PROGRAM P_StationOpenLock
VAR
	_station:					REFERence TO ST_SystemStation;
	_bEnable: 					BOOL;
	_OpenLockCheck0FTrig:       Tc2_Standard.F_TRIG;
END_VAR

_station REF= G_arrStation[E_Station.OpenLock];
_station.arrName[E_Language.Chinese]:="解锁站";
_station.arrName[E_Language.Vietnamese]:="Mở khóa nhà ga";
_bEnable:=NOT GVL.stSetting.arrStationShield[E_Station.OpenLock];

IF GVL_Data.stRecipe.eMachineType=E_MachineType._311 THEN
	A_Home311();
	A_Auto311();
ELSE
	A_Home();
	A_Auto();
END_IF

_OpenLockCheck0FTrig(CLK:= GVL.I.bOpenLockCheck0, Q=> );

GVL._arrAutoTimer[E_Timer.SteeringCheck1F](IN:=NOT GVL.I.bSteeringCheck1 AND GVL.I.bSteeringAcquireElevator_Cyl_H, PT:=TO_TIME(GVL_Data.stRecipe.arrAutoTon[E_Timer.SteeringCheck1F]), Q=>GVL._arrAutoTimerOut[E_Timer.SteeringCheck1F] , ET=> );

ACTION A_Auto:
CASE _station.iStepNow OF
	1000:
		_station.arrInfo[E_Language.Chinese]:="初始化完成等待启动";
		IF _bEnable THEN
			_station.iStepNext:=1101;
		END_IF
	1101:
		_station.arrInfo[E_Language.Chinese]:="判断是否有料";
		IF NOT GVL.I.bOpenLockCheck THEN
			_station.iStepNext:=1201;
		END_IF
	1201:
		_station.arrInfo[E_Language.Chinese]:="请求上料";
		GVL.stHandshake.bOpenToSteering:=TRUE;
		IF GVL.stHandshake.bSteeringToOpen THEN
			_station.iStepNext:=1301;
		END_IF
	1301:
		_station.arrInfo[E_Language.Chinese]:="等待产品从旋转站流出";
		GVL.stOverTime.bOpenLockCheck:=TRUE;
		IF GVL._arrAutoTimerOut[E_Timer.SteeringCheck1F] THEN
			GVL.stOverTime.bOpenLockCheck:=FALSE;
			_station.iStepNext:=1401;//解锁站流入传感器安装后改为 1311
		END_IF
	1311:		
		_station.arrInfo[E_Language.Chinese]:="产品从旋转站流出确认";
		IF _OpenLockCheck0FTrig.Q THEN
			_station.iStepNext:=1401;
		END_IF	
	1401:
		_station.arrInfo[E_Language.Chinese]:="复位上料请求";
		GVL.stHandshake.bOpenToSteering:=FALSE;
		IF  NOT GVL.stHandshake.bSteeringToOpen THEN
			_station.iStepNext:=1411;
		END_IF
	1411:
		_station.arrInfo[E_Language.Chinese]:="等待产品到位";
		GVL.stOverTime.bOpenLockCheck:=TRUE;
		IF GVL.I.bOpenLockCheck THEN
			GVL.stOverTime.bOpenLockCheck:=FALSE;
			_station.iStepNext:=1501;
		END_IF			
	1501:
		_station.arrInfo[E_Language.Chinese]:="顶升气缸伸出";
		IF G_arrFbCylinder[E_Cylinder.OpenLockLift].M_WorkRequest() THEN
			IF GVL_Data.stRecipe.eMachineType=E_MachineType._373 AND NOT GVL.stSetting.bOpenLockPressShield THEN 
				_station.iStepNext:=1511;
			ELSE
			_station.iStepNext:=1601;
			END_IF
		END_IF
	1511:	
		_station.arrInfo[E_Language.Chinese]:="解压侧推气缸伸出";	
		IF G_arrFbCylinder[E_Cylinder.OpenLockPressPush].M_WorkRequest() THEN
			_station.iStepNext:=1521;
		END_IF
	1521:	
		_station.arrInfo[E_Language.Chinese]:="解压旋转气缸旋转";	
		IF G_arrFbCylinder[E_Cylinder.OpenLockPressRotate].M_WorkRequest() THEN
			_station.iStepNext:=1531;
		END_IF	
	1531:	
		_station.arrInfo[E_Language.Chinese]:="解压旋转气缸返回";	
		IF G_arrFbCylinder[E_Cylinder.OpenLockPressRotate].M_HomeRequest() THEN
			_station.iStepNext:=1541;		
		END_IF		
	1541:
		_station.arrInfo[E_Language.Chinese]:="解压侧推气缸缩回 侧推气缸伸出";
		IF M_PushWork() AND G_arrFbCylinder[E_Cylinder.OpenLockPressPush].M_HomeRequest() THEN
			_station.iStepNext:=1701;
		END_IF		
	1601:
		_station.arrInfo[E_Language.Chinese]:="侧推气缸伸出";
		IF M_PushWork() THEN
			_station.iStepNext:=1701;
		END_IF
	1701:
		_station.arrInfo[E_Language.Chinese]:="旋转气缸至右位 校平气缸伸出";
		IF G_arrFbCylinder[E_Cylinder.OpenLockRotate].M_WorkRequest() AND M_StandardWork() THEN
			_station.iStepNext:=1801;
		END_IF
	1801:
		_station.arrInfo[E_Language.Chinese]:="侧推气缸缩回 校平气缸缩回 阻挡气缸缩回";
		IF M_PushHome() AND M_StandardHome()  AND  G_arrFbCylinder[E_Cylinder.OpenLockPrevent].M_HomeRequest() THEN
           _station.iStepNext:=2001;
		END_IF
	2001:
		_station.arrInfo[E_Language.Chinese]:="等待取Uc站请求放料";
		IF GVL.stHandshake.bTakeUcToOpen THEN
			GVL.stHandshake.bOpenToTakeUc:=TRUE;
			GVL.stHandshake.bOpenToSteering:=TRUE;//同时请求旋转站放料
			_station.iStepNext:=2101;
		END_IF
	2101:
	     _station.arrInfo[E_Language.Chinese]:="顶升气缸下降,解锁旋转气缸至左位";
		IF G_arrFbCylinder[E_Cylinder.OpenLockLift].M_HomeRequest() AND G_arrFbCylinder[E_Cylinder.OpenLockRotate].M_HomeRequest() THEN
			_station.iStepNext:=2201;
		END_IF
	2201:
		_station.arrInfo[E_Language.Chinese]:="等待复位请求信号";
		IF NOT GVL.stHandshake.bTakeUcToOpen THEN
			GVL.stHandshake.bOpenToTakeUc:=FALSE;
			_station.iStepNext:=2301;
		END_IF		
	2301:
		_station.arrInfo[E_Language.Chinese]:="阻挡气缸伸出";
		IF G_arrFbCylinder[E_Cylinder.OpenLockPrevent].M_WorkRequest() THEN
			_station.iStepNext:=1201;
		END_IF		

END_CASE
END_ACTION

ACTION A_Auto311:
CASE _station.iStepNow OF
	1000:
		_station.arrInfo[E_Language.Chinese]:="初始化完成等待启动";
		IF _bEnable THEN
			_station.iStepNext:=1101;
		END_IF
	1101:
		_station.arrInfo[E_Language.Chinese]:="判断是否有料";
		IF NOT GVL.I.bOpenLockCheck THEN
			_station.iStepNext:=1201;
		END_IF
	1201:
		_station.arrInfo[E_Language.Chinese]:="请求上料";
		GVL.stHandshake.bOpenToSteering:=TRUE;
		IF GVL.stHandshake.bSteeringToOpen THEN
			_station.iStepNext:=1301;
		END_IF
	1301:
		_station.arrInfo[E_Language.Chinese]:="等待产品从旋转站流出";
		GVL.stOverTime.bOpenLockCheck:=TRUE;
		IF GVL._arrAutoTimerOut[E_Timer.SteeringCheck1F] THEN
			GVL.stOverTime.bOpenLockCheck:=FALSE;
			_station.iStepNext:=1401;//传感器安装后改为 1311
		END_IF
	1311:		
		_station.arrInfo[E_Language.Chinese]:="产品从旋转站流出确认";
		IF _OpenLockCheck0FTrig.Q THEN
			_station.iStepNext:=1401;
		END_IF			
	1401:
		_station.arrInfo[E_Language.Chinese]:="复位上料请求";
		GVL.stHandshake.bOpenToSteering:=FALSE;
		IF  NOT GVL.stHandshake.bSteeringToOpen THEN
			_station.iStepNext:=1411;
		END_IF
	1411:
		_station.arrInfo[E_Language.Chinese]:="等待产品到位";
		GVL.stOverTime.bOpenLockCheck:=TRUE;
		IF GVL.I.bOpenLockCheck THEN
			GVL.stOverTime.bOpenLockCheck:=FALSE;
			_station.iStepNext:=1501;
		END_IF			
	1501:
		_station.arrInfo[E_Language.Chinese]:="顶升气缸伸出";
		IF G_arrFbCylinder[E_Cylinder.OpenLockLift].M_WorkRequest() THEN
			_station.iStepNext:=1511;
		END_IF
	1511:		
		_station.arrInfo[E_Language.Chinese]:="检测工装有无误合盖";
		IF GVL.I.bFrockCloseCheck OR GVL.stSetting.bFrockCloseCheckShield THEN
			_station.iStepNext:=1601;
		ELSE
			_station.iStepNext:=1521;
		END_IF
	1521:	
		_station.arrInfo[E_Language.Chinese]:="置位工装检测失败记忆";
		GVL.TakeUcSafeCheckNG_OpenLock:=TRUE;
		IF GVL.TakeUcSafeCheckNG_OpenLock THEN
			_station.iStepNext:=2001;
		END_IF		
	1601:
		_station.arrInfo[E_Language.Chinese]:="升降气缸缩回";
		GVL.TakeUcSafeCheckNG_OpenLock:=FALSE;
		IF G_arrFbCylinder[E_Cylinder.OpenLockElevator].M_HomeRequest() THEN
			_station.iStepNext:=1701;
		END_IF
	1701:
		_station.arrInfo[E_Language.Chinese]:="按压气缸伸出";
		IF G_arrFbCylinder[E_Cylinder.OpenLockPin].M_WorkRequest() THEN
			_station.iStepNext:=1801;
		END_IF
	1801:
		_station.arrInfo[E_Language.Chinese]:="平移气缸缩回";
		IF G_arrFbCylinder[E_Cylinder.OpenLockTranslation].M_HomeRequest() THEN
			_station.iStepNext:=1901;
		END_IF
	1901:
		_station.arrInfo[E_Language.Chinese]:="旋转气缸至初始位";
		IF G_arrFbCylinder[E_Cylinder.OpenLockRotate].M_HomeRequest() THEN
			_station.iStepNext:=1951;
		END_IF
	1951:
		_station.arrInfo[E_Language.Chinese]:="升降气缸伸出 按压气缸缩回";
		IF G_arrFbCylinder[E_Cylinder.OpenLockElevator].M_WorkRequest() AND G_arrFbCylinder[E_Cylinder.OpenLockPin].M_HomeRequest()  THEN
			_station.iStepNext:=2001;
		END_IF
	2001:
		_station.arrInfo[E_Language.Chinese]:="等待取Uc站请求放料";
		IF GVL.stHandshake.bTakeUcToOpen THEN
			GVL.stHandshake.bOpenToTakeUc:=TRUE;
			GVL.stHandshake.bOpenToSteering:=TRUE;//同时请求旋转站放料
			_station.iStepNext:=2051;
		END_IF
	2051:
		_station.arrInfo[E_Language.Chinese]:="顶升气缸缩回 阻挡气缸缩回";
		IF G_arrFbCylinder[E_Cylinder.OpenLockPrevent].M_HomeRequest() AND G_arrFbCylinder[E_Cylinder.OpenLockLift].M_HomeRequest() THEN
			_station.iStepNext:=2101;
		END_IF
	2101:
		_station.arrInfo[E_Language.Chinese]:="旋转气缸至工作位 平移气缸伸出";
		G_arrFbCylinder[E_Cylinder.OpenLockRotate].M_WorkRequest();
		G_arrFbCylinder[E_Cylinder.OpenLockTranslation].M_WorkRequest();
		_station.iStepNext:=2201;		
	2201:
		_station.arrInfo[E_Language.Chinese]:="等待复位请求信号";
		IF NOT GVL.stHandshake.bTakeUcToOpen THEN
			GVL.stHandshake.bOpenToTakeUc:=FALSE;
			_station.iStepNext:=2301;
		END_IF
	2301:
		_station.arrInfo[E_Language.Chinese]:="阻挡气缸伸出";
		IF G_arrFbCylinder[E_Cylinder.OpenLockPrevent].M_WorkRequest() AND G_arrFbCylinder[E_Cylinder.OpenLockRotate].M_WorkRequest() AND G_arrFbCylinder[E_Cylinder.OpenLockTranslation].M_WorkRequest() THEN
			_station.iStepNext:=1201;
		END_IF

END_CASE
END_ACTION

ACTION A_Home:
CASE _station.iStepNow OF
	0:
		_station.arrInfo[E_Language.Chinese]:="等待初始化";
		_station.iStepNext:=SEL(_bEnable,1000,100);
	100:		
		IF GVL_Data.stRecipe.eMachineType=E_MachineType._373 AND NOT GVL.stSetting.bOpenLockPressShield THEN 
			_station.iStepNext:=110;
		ELSE
			_station.iStepNext:=150;
		END_IF		
	110:
		_station.arrInfo[E_Language.Chinese]:="解压旋转气缸返回";
		IF G_arrFbCylinder[E_Cylinder.OpenLockPressRotate].M_HomeRequest() THEN
			_station.iStepNext:=120;
		END_IF	
	120:
		_station.arrInfo[E_Language.Chinese]:="解压侧推气缸缩回";
		IF G_arrFbCylinder[E_Cylinder.OpenLockPressPush].M_HomeRequest() THEN
			_station.iStepNext:=150;
		END_IF	
	150:	
		_station.arrInfo[E_Language.Chinese]:="侧推气缸缩回";
		IF M_PushHome() THEN
			_station.iStepNext:=200;
		END_IF
	200:
		_station.arrInfo[E_Language.Chinese]:="旋转气缸至左位";
		IF G_arrFbCylinder[E_Cylinder.OpenLockRotate].M_HomeRequest() THEN
			_station.iStepNext:=300;
		END_IF
	300:
		_station.arrInfo[E_Language.Chinese]:="阻挡气缸伸出";
		IF G_arrFbCylinder[E_Cylinder.OpenLockPrevent].M_WorkRequest() THEN
			_station.iStepNext:=400;
		END_IF
	400:
		_station.arrInfo[E_Language.Chinese]:="顶升气缸缩回";
		IF G_arrFbCylinder[E_Cylinder.OpenLockLift].M_HomeRequest() THEN
			_station.iStepNext:=500;
		END_IF
	500:
		_station.arrInfo[E_Language.Chinese]:="校平气缸缩回";
		IF  M_StandardHome() THEN
			_station.iStepNext:=1000;
		END_IF
END_CASE
END_ACTION

ACTION A_Home311:
CASE _station.iStepNow OF
	0:
		_station.arrInfo[E_Language.Chinese]:="等待初始化";
		_station.iStepNext:=SEL(_bEnable,1000,100);
	100:
		_station.arrInfo[E_Language.Chinese]:="升降气缸伸出";
		IF 	G_arrFbCylinder[E_Cylinder.OpenLockElevator].M_WorkRequest() THEN
			_station.iStepNext:=150;
		END_IF
	150:
		_station.arrInfo[E_Language.Chinese]:="按压气缸缩回";
		IF G_arrFbCylinder[E_Cylinder.OpenLockPin].M_HomeRequest() THEN
			_station.iStepNext:=200;
		END_IF
	200:
		_station.arrInfo[E_Language.Chinese]:="旋转气缸至工作位";
		IF G_arrFbCylinder[E_Cylinder.OpenLockRotate].M_WorkRequest() THEN
			_station.iStepNext:=300;
		END_IF
	300:
		_station.arrInfo[E_Language.Chinese]:="平移气缸伸出";
		IF 	G_arrFbCylinder[E_Cylinder.OpenLockTranslation].M_WorkRequest() THEN
			_station.iStepNext:=500;
		END_IF
	500:
		_station.arrInfo[E_Language.Chinese]:="阻挡气缸伸出";
		IF G_arrFbCylinder[E_Cylinder.OpenLockPrevent].M_WorkRequest() THEN
			_station.iStepNext:=600;
		END_IF
	600:
		_station.arrInfo[E_Language.Chinese]:="顶升气缸缩回";
		IF G_arrFbCylinder[E_Cylinder.OpenLockLift].M_HomeRequest() THEN
			_station.iStepNext:=1000;
		END_IF
END_CASE
END_ACTION

METHOD M_PushHome : BOOL
VAR_INPUT
END_VAR
CASE GVL_Data.stRecipe.eMachineType OF
	E_MachineType._200,E_MachineType._069,E_MachineType._367:
		M_PushHome:=G_arrFbCylinder[E_Cylinder.OpenLockPush].M_HomeRequest() AND G_arrFbCylinder[E_Cylinder.OpenLockPush2].M_HomeRequest();
	E_MachineType._373:
		M_PushHome:=G_arrFbCylinder[E_Cylinder.OpenLockPush].M_HomeRequest();
END_CASE
END_METHOD

METHOD M_PushWork : BOOL
VAR_INPUT
END_VAR
CASE GVL_Data.stRecipe.eMachineType OF
	E_MachineType._200,E_MachineType._069,E_MachineType._367:
		M_PushWork:=G_arrFbCylinder[E_Cylinder.OpenLockPush].M_WorkRequest() AND G_arrFbCylinder[E_Cylinder.OpenLockPush2].M_WorkRequest();
	E_MachineType._373:
		M_PushWork:=G_arrFbCylinder[E_Cylinder.OpenLockPush].M_WorkRequest();
END_CASE
END_METHOD

METHOD M_StandardHome : BOOL
VAR_INPUT
END_VAR
M_StandardHome:=TRUE;
END_METHOD

METHOD M_StandardWork : BOOL
VAR_INPUT
END_VAR
M_StandardWork:=TRUE;
END_METHOD

END_PROGRAM

(* stored: Version 1.1.0.1, ProductVersion 3.1.4024.3
   POU P_StationOpenLock: Id {ce5dff6b-fe73-4149-9003-dba4a98bca8a}, SpecialFunc None
   Action A_Auto: Id {e584a16f-aecc-45a3-861e-dc548a74eb21}
   Action A_Auto311: Id {e2bc8e2f-b230-45d3-a820-67c85b360fc4}
   Action A_Home: Id {259e29a1-5d1d-409a-97b0-e3ba595953c7}
   Action A_Home311: Id {f41d7e3f-f59d-4a11-b2a3-ff6cd046e966}
   Method M_PushHome: Id {247571e8-b315-4ace-b90e-bd4738cabec3}
   Method M_PushWork: Id {4ca4089a-fc2f-42be-8a15-dc9f90c2db48}
   Method M_StandardHome: Id {259da1d9-d1e5-4801-898e-5e889d2b5202}
   Method M_StandardWork: Id {4acf037f-b781-4646-bdd1-e69cf1e0d70a} *)
